(*			
	RAFALOS
	Rafał Osajda		19.09.2025		TC 4024.66
	Rodzic dla wszystkich elementów wykonawczych
*)
FUNCTION_BLOCK FB_BaseExecutiveElement EXTENDS FB_BaseComponent IMPLEMENTS ITF_BaseExecutiveElement
VAR
END_VAR

END_FUNCTION_BLOCK

(* stored: Version 1.1.0.1
   POU FB_BaseExecutiveElement: Id {4411e8b6-2e2c-0151-1419-8a5f32f7c37c}, SpecialFunc None *)
